TYPE ST_EM_Cmd_UpdateTable :
	STRUCT
		ChangeTable : BOOL;
		ChangeMode	: BOOL;
	END_STRUCT
END_TYPE

(* stored: Version 1.1.0.1
   DUT ST_EM_Cmd_UpdateTable: Id {cd279b59-7dad-41d5-b05a-803600e3de62} *)
